FUNCTION_BLOCK FB_VGC_Test EXTENDS TcUnit.FB_TestSuite
VAR_INPUT
END_VAR
VAR_OUTPUT
END_VAR
VAR
    VGC: FB_VGC;
    US_IG : ST_VG;
    DS_IG : ST_VG;
    io_fbFFHWO    :    FB_HardwareFFOutput;
    TotalTests : INT:=0;
    ex               : __SYSTEM.ExceptionCode;
END_VAR

M_INIT();
M_Interlock();

METHOD M_Check_State
VAR_INPUT
END_VAR
END_METHOD

METHOD M_INIT : BOOL
VAR//_INPUT

END_VAR
TEST('VGC_Startup');
This^.US_IG.rPRESS := 1E-9;
This^.US_IG.xPRESS_OK := TRUE;
This^.US_IG.xAT_VAC := TRUE;

This^.DS_IG.rPRESS := 1E-9;
This^.DS_IG.xPRESS_OK := TRUE;

(*This^.VGC(
    i_stUSG:= This^.US_IG,
    i_stDSG:= This^.DS_IG ,
    i_xDis_DPIlk:= FALSE,
    i_xEPS_OK:= TRUE ,
    //i_xPMPS_OK:= TRUE,
    i_xExt_OK:= TRUE,
    i_xOverrideMode:= ,
    i_xReset:= ,
    iq_stValve=> ,
    xMPS_OK=> ,
    io_fbFFHWO:= This^.io_fbFFHWO,
    fbArbiter:=g_fbArbiter);
*)
AssertFalse(This^.VGC.iq_stValve.pv_xOPN_SW,'VGC pv_xOPN_SW is set to true');
AssertFalse(VGC.iq_stValve.q_xOPN_DO,'VGC q_xOPN_DO is set to true');
TEST_FINISHED_NAMED('VGC_Startup');
END_METHOD

METHOD M_Interlock : BOOL
VAR//_INPUT

END_VAR
// Test interlock is active and attempting to open valve
TEST('VGC_Interlock_Active');
This^.US_IG.xPRESS_OK := FALSE;
This^.DS_IG.xPRESS_OK := FALSE;
VGC.M_Set_OPN_SW(TRUE);
// run the function block one more time
(*VGC(
    i_stUSG:= US_IG,
    i_stDSG:= DS_IG ,
    i_xDis_DPIlk:= FALSE,
    i_xEPS_OK:= TRUE ,
    i_xPMPS_OK:= TRUE ,
    i_xExt_OK:= TRUE,
    i_xOverrideMode:= ,
    i_xReset:= ,
    iq_stValve=> ,
    xMPS_OK=> ,
    io_fbFFHWO:= io_fbFFHWO);*)
AssertFalse(VGC.iq_stValve.pv_xOPN_SW,'VGC pv_xOPN_SW is set to true');
AssertFalse(VGC.iq_stValve.q_xOPN_DO,'VGC q_xOPN_DO is set to true');
TEST_FINISHED_NAMED('VGC_Interlock_Active');
// Test interlock is not active and attempting to open valve
TEST('VGC_Interlock_OK');
This^.US_IG.xPRESS_OK := TRUE;
This^.DS_IG.xPRESS_OK := TRUE;
VGC.M_Set_OPN_SW(TRUE);
// run the function block one more time
(*VGC(
    i_stUSG:= US_IG,
    i_stDSG:= DS_IG ,
    i_xDis_DPIlk:= FALSE,
    i_xEPS_OK:= ,
    i_xPMPS_OK:= ,
    i_xExt_OK:= ,
    i_xOverrideMode:= ,
    i_xReset:= ,
    iq_stValve=> ,
    xMPS_OK=> ,
    io_fbFFHWO:= io_fbFFHWO);*)
AssertTrue(VGC.iq_stValve.pv_xOPN_SW,'VGC pv_xOPN_SW is set to false');
AssertTrue(VGC.iq_stValve.q_xOPN_DO,'VGC q_xOPN_DO is set to false');
TEST_FINISHED_NAMED('VGC_Interlock_OK');
// Test interlock ok lost while valve is open
TEST('VGC_Interlock_Lost');
This^.US_IG.xPRESS_OK := False;
This^.DS_IG.xPRESS_OK := TRUE;
// run the function block one more time
(*VGC(
    i_stUSG:= US_IG,
    i_stDSG:= DS_IG ,
    i_xDis_DPIlk:= FALSE,
    i_xEPS_OK:= ,
    i_xPMPS_OK:= ,
    i_xExt_OK:= ,
    i_xOverrideMode:= ,
    i_xReset:= ,
    iq_stValve=> ,
    xMPS_OK=> ,
    io_fbFFHWO:= io_fbFFHWO);*)
AssertFalse(VGC.iq_stValve.pv_xOPN_SW,'VGC pv_xOPN_SW is set to true');
AssertFalse(VGC.iq_stValve.q_xOPN_DO,'VGC q_xOPN_DO is set to true');
TEST_FINISHED_NAMED('VGC_Interlock_Lost');
END_METHOD

END_FUNCTION_BLOCK

(* stored: Version 1.1.0.1
   POU FB_VGC_Test: Id {f7068602-850f-4f85-937b-c57c62973b92}, SpecialFunc None
   Method M_Check_State: Id {323f8a43-3288-4a88-896a-0ee6bf963246}
   Method M_INIT: Id {872ba40e-8e0d-4855-ae6d-7645f3617e36}
   Method M_Interlock: Id {35580cdf-b62c-4fb5-b5f0-7ced6771af19} *)
